(* PLC project creation, Dassault Systèmes ControlBuild 2024x *)
(* stored: creationDateTime 2023-10-03T11:13:55-01:00 *)

FUNCTION_BLOCK tri_chain.creation
  VAR_OUTPUT
    idProd : DINT := 0;
    creationFailed : BOOL := false;
  END_VAR
  VAR
    status_act_prod : DINT := 0;
    m11 : REAL := 1.0;
    m12 : REAL := 0.0;
    m13 : REAL := 0.0;
    m14 : REAL := 0.0;
    m21 : REAL := 0.0;
    m22 : REAL := 1.0;
    m23 : REAL := 0.0;
    m24 : REAL := 0.0;
    m31 : REAL := 0.0;
    m32 : REAL := 0.0;
    m33 : REAL := 1.0;
    m34 : REAL := 0.0;
    m41 : REAL := 0.0;
    m42 : REAL := 0.0;
    m43 : REAL := 0.0;
    m44 : REAL := 1.0;
    px : REAL := 0.0;
    py : REAL := 0.0;
    pz : REAL := 0.0;
    dx : REAL := 0.0;
    dy : REAL := 0.0;
    dz : REAL := 0.0;
    presenceProduct : BOOL := false;
    arrival_PB : BOOL := false;
    time2reach : REAL := 0.0;
    edge_arrival_PB : BOOL := false;
    first : BOOL := true;
  END_VAR
  VAR CONSTANT
    pulseType : BOOL := false;
    pulseDuration : REAL := 10.0;
  END_VAR


ACTION C_source_code:
/* ----------------------------------------------------------------	*/
/* Type : Model of Operative Behaviour					*/
/* Category :  Product							*/
/* Author : Dassault Systemes						*/
/* Update date : June 2018							*/
/* ----------------------------------------------------------------	*/
/* This module simulates the arrival of work pieces in a plant.	*/
/*	The actor cretaes a product when the user acts on a		*/
/*	launching push-button					.	*/
/* -----------------------------------------------------------------	*/
if(first) {
	edge_arrival_PB = arrival_PB;
	first = 0;
}

if pulseType {
	if arrival_PB{
		if(timeNow >= time2reach) arrival_PB=0;
	}else {
		time2reach = timeNow + (pulseDuration * 1000000);
	}
} else {
	if((edge_arrival_PB < arrival_PB) || (edge_arrival_PB > arrival_PB)){
		time2reach = timeNow + (pulseDuration * 1000000);
	}  else {
		if(timeNow >= time2reach) arrival_PB = ! arrival_PB;
	}
}

if ((edge_arrival_PB < arrival_PB) && ! presenceProduct) {
	idProd=prodNew(tri_chain__boxtri,px,py,pz,dx,dy,dz);
	if(idProd < 0) creationFailed = 1;
}

presenceProduct=0;

edge_arrival_PB = arrival_PB;
END_ACTION

ACTION C_header:
#include "tri_chain/functional/boxtri/boxtri.h"
END_ACTION
END_FUNCTION_BLOCK
